FUNCTION_BLOCK ABSTRACT FB_Abstract_FunktionCtrl IMPLEMENTS I_FunctionCtrl
VAR_INPUT
END_VAR
VAR_OUTPUT
END_VAR
VAR
END_VAR

{warning 'Eigenschaftenimplementierung hinzufügen'}
PROPERTY Busy : BOOL
GET
END_GET
END_PROPERTY

{warning 'Eigenschaftenimplementierung hinzufügen'}
PROPERTY Done : BOOL
GET
END_GET
END_PROPERTY

{warning 'Eigenschaftenimplementierung hinzufügen'}
PROPERTY Error : BOOL
GET
END_GET
END_PROPERTY

{warning 'Eigenschaftenimplementierung hinzufügen'}
PROPERTY ErrorCode : WORD
GET
END_GET
END_PROPERTY

{warning 'Methodenimplementierung hinzufügen'}
METHOD Execute : BOOL
END_METHOD

{warning 'Eigenschaftenimplementierung hinzufügen'}
PROPERTY Ready : BOOL
GET
END_GET
END_PROPERTY

{warning 'Methodenimplementierung hinzufügen'}
METHOD Reset : BOOL
END_METHOD

END_FUNCTION_BLOCK

(* stored: Version 1.1.0.1, ProductVersion 3.1.4024.12
   POU FB_Abstract_FunktionCtrl: Id {ff5f2b89-1b30-43c2-a00b-c8ec90b43ee8}, SpecialFunc None
   Property Busy: Id {497c1c79-67ce-475a-a452-b4670b01db12}
   Get Get: Id {b8b4f636-0d4a-408d-97de-2e9401191a01}
   Property Done: Id {a0f4a82f-3362-40ab-90a0-0011c210bc70}
   Get Get: Id {adae057c-2684-42b9-a198-2d01bde115a5}
   Property Error: Id {4330901d-d320-480e-9eb4-59415bbc5581}
   Get Get: Id {bcbe9b96-a283-4c08-8b70-63d7ce4a14ea}
   Property ErrorCode: Id {0eb279b9-0427-4070-a0a0-71d3fda85eb2}
   Get Get: Id {6abf26f8-7f80-4879-bd81-1fe656a46730}
   Method Execute: Id {e0d3cf87-10e2-4494-88e5-b0c097c56d1b}
   Property Ready: Id {2840f109-1265-47cc-9854-00cdd2edf4b0}
   Get Get: Id {8598d7ce-0e7d-4f71-8bc4-31055f4d134d}
   Method Reset: Id {ed6deedd-244e-40eb-9e89-ef9e83a462d9} *)
